INTERFACE PUBLIC ClearingCommands EXTENDS ClearedStateCommands, ActionStateCommands

END_INTERFACE

(* stored: Version 1.1.0.1, ProductVersion 3.1.4026.18
   Itf ClearingCommands: Id {e5c1cdf7-471e-0292-28be-8a8a5b1d0479} *)
